// TwinCAT 3 PLC project hydValve
// ProgramVersion: 3.1.4024.0
// libraries:
//   Tc2_Standard, * (Beckhoff Automation GmbH)
//   Tc2_System, * (Beckhoff Automation GmbH)
//   Tc3_Module, * (Beckhoff Automation GmbH)
// project tree:
//   DUTs/ configaracionParammetrs.TcDUT, Staus.TcDUT
//   GVLs/ generalVariable.TcGVL
//   / PlcTask.TcTTO
//   POUs/ accelerationValve.TcPOU, blockMessage.TcPOU, decelerationValve.TcPOU, MAIN.TcPOU, Valve.TcPOU
// real-time tasks:
//   TASK PlcTask: cycle T#10ms, priority 20, ADS port 350

CONFIGURATION hydValve
    RESOURCE PLC ON TwinCAT3
        TASK PlcTask(INTERVAL := T#10ms, PRIORITY := 20);
        PROGRAM MAIN WITH PlcTask : MAIN;
    END_RESOURCE
END_CONFIGURATION

// ---- DUTs/configaracionParammetrs.TcDUT
TYPE configaracionParammetrs :
STRUCT
	CurPosDirMin : REAL := 100; // Minimální proud na solenoid v daném směru [mA]
	CurPosDirMax : REAL := 500; // Maximální proud na solenoid v daném směru [mA]
	CurNegDirMin : REAL := 100; // Minimální proud na solenoid v daném směru [mA]
	CurNegDirMax : REAL := 500; // Maximální proud na solenoid v daném směru [mA]
	RampPosDirUp : INT := 100; // Doba změny z min. na max. otevření v daném směru [ms]
	RampPosDirDown :INT := 100; // Doba změny z max. na min. otevření v daném směru [ms]
	RampNegDirUp : INT := 100; // Doba změny z min. na max. otevření v daném směru [ms]
	RampNegDirDown : INT := 100; // Doba změny z max. na min. otevření v daném směru [ms]
	Deadtime : INT := 5; // Kompenzace setrvačnosti při reverzaci [ms]

END_STRUCT
END_TYPE

// ---- DUTs/Staus.TcDUT
TYPE Staus :
STRUCT
	Standstill : BOOL;	// Oba výstupy jsou na minimu
	Accel : BOOL;	// Jeden z výstupů zrychluje
	Decel : BOOL;	// Jeden z výstupů zpomaluje
	OutPosDirProc : REAL;// Výstup v daném směru [%]
	OutNegDirProc : REAL;// Výstup v daném směru [%]
	bBussy : BOOL;// TRUE je-li FB aktivní (změna na výstupu)
	bDone : BOOL;	// TRUE je-li výstupní hodnota je rovna žádané
	bError : STRING; // Chyba
	nErrorId : INT;// Kód chyby
END_STRUCT
END_TYPE

// ---- GVLs/generalVariable.TcGVL
{attribute 'qualified_only'}
VAR_GLOBAL
	conParammetr : configaracionParammetrs;
	staus : Staus;
END_VAR

// ---- POUs/MAIN.TcPOU
PROGRAM MAIN
VAR
	
	hydraulicValve : Valve;
	enaNegDirB : BOOL := FALSE;
	enaPosDirB : BOOL := FALSE;
	commandSet : REAL := 0;
	//konfiguraParametry : REFERENCE TO configaracionParammetrs  REF=generalVariable.conParammetr;
	OutPosDir : REAL := 0 ;	// Výstup v daném směru [mA]
	OutNegDir : REAL := 0 ;	// Výstup v daném směru [mA]
END_VAR


//hydraulicValve.configaracionParammetr := generalVariable.conParammetr;

hydraulicValve.enableSolenoidControl(poz :=enaPosDirB, neg := enaNegDirB);
hydraulicValve.commandCheck(commandSet);
hydraulicValve();
OutNegDir := hydraulicValve.OutNegDir;
OutPosDir := hydraulicValve.OutPosDir;

END_PROGRAM

// ---- POUs/Valve.TcPOU
FUNCTION_BLOCK Valve
VAR_INPUT
	//configaracionParammetr : configaracionParammetrs;
END_VAR
VAR		
	
	enaNegDir : BOOL := FALSE;
	enaPosDir : BOOL := FALSE;
	command : REAL; // Příkaz -1000 .. 0 .. 1000 [procenta * 10]

	errorDir : BOOL;
	
	currentCommand : REAL := 0;
	prolaz : STRING;
	previousenaNegDir : BOOL; 
	previousenaPosDir : BOOL;
	currentError : BOOL := FALSE; // test error
	
	//command : INT; 
	status : REFERENCE TO Staus REF=generalVariable.staus;
	konfiguraParametry : REFERENCE TO configaracionParammetrs  REF=generalVariable.conParammetr;
	speedRamp : REAL;
	mAcurrentCommand : REAL; 
	mAcommand : REAL;
END_VAR
VAR_OUTPUT
	OutPosDir : REAL := 0 ;	// Výstup v daném směru [mA]
	OutNegDir : REAL := 0 ;	// Výstup v daném směru [mA]
END_VAR

//currentDir := currentDirB(enaNegDir,enaPosDir);
mAcurrentCommand := convertToAnal(ABS(currentCommand*10));
mAcommand :=  convertToAnal(ABS(command*10));

IF (currentCommand = 0) THEN
	OutNegDir := mAcurrentCommand;
	OutPosDir := mAcurrentCommand;
	waitbDeathtime();
	ELSIF enaPosDir > 0 THEN
		OutPosDir := mAcurrentCommand;
		OutNegDir := convertToAnal(0);
		ELSE
			OutNegDir := mAcurrentCommand;
			OutPosDir := convertToAnal(0);
	END_IF;

signalStandstill();
prolaz := 'fb';
IF (currentcommand <> command) THEN
		//nTime := elapsTime(direction := currentDir);
		prolaz := 'različiti';
		currentcommand := rampValve ();
	ELSE	
		Accel_Decel(FALSE, FALSE);
		status.bDone := TRUE;
END_IF;

METHOD PRIVATE Accel_Decel
VAR_INPUT
	a : BOOL;
	b : BOOL;
END_VAR
status.Accel := a;
status.Decel := b;
END_METHOD

METHOD addCommand
VAR_INPUT
	comm : real;
END_VAR
command := comm;	
currentError := FALSE;
errorDir := FALSE;
END_METHOD

METHOD PUBLIC commandCheck
VAR_INPUT
	comm : REAL;
END_VAR
VAR
	
END_VAR
IF not(currentError) THEN
	IF ((comm <= 100) AND (comm >0)) THEN
			IF enaPosDir THEN
				addCommand(comm);
			ELSIF NOT(errorDir) THEN
					errCode(4);
					errorDir := TRUE;
				END_IF
		ELSIF ((comm >= -100) AND (comm < 0)) THEN
				IF enaNegDir THEN
					addCommand(comm);
				ELSIF not(errorDir) THEN
					errCode(3);
					errorDir := TRUE;
				END_IF
				ELSIF comm = 0 THEN
						status.Standstill := 0;
						addCommand(comm);
					ELSIF NOT(errorDir) THEN
					errCode(2);
					errorDir := TRUE;
				END_IF
END_IF
END_METHOD

METHOD PRIVATE convertTo : REAL
VAR_INPUT
	currCommand : REAL;
END_VAR
IF enaPosDir THEN
	convertTo := 100*(currCommand -konfiguraParametry.CurPosDirMin)/(konfiguraParametry.CurPosDirMax - konfiguraParametry.CurPosDirMin);
ELSE
	convertTo := 100*(currCommand -konfiguraParametry.CurNegDirMin)/(konfiguraParametry.CurnegDirMax - konfiguraParametry.CurNegDirMin);
END_IF
END_METHOD

METHOD PROTECTED convertToAnal : REAL
VAR_INPUT
	pCommand : REAL;
END_VAR
IF  enaPosDir THEN
	convertToAnal:= (pCommand * (konfiguraParametry.CurPosDirMax - konfiguraParametry.CurPosDirMin)/1000) + konfiguraParametry.CurPosDirMin;
ELSE
	convertToAnal:= (pCommand * (konfiguraParametry.CurNegDirMax - konfiguraParametry.CurNegDirMin)/1000) + konfiguraParametry.CurNegDirMin;
END_IF
END_METHOD

METHOD PRIVATE elapsTime : REAL
VAR_INPUT
	direction : BOOL;
END_VAR
IF direction THEN
		elapsTime := (konfiguraParametry.CurPosDirMax - konfiguraParametry.CurPosDirMin)/(konfiguraParametry.RampPosDirDown -konfiguraParametry.RampPosDirUp);
	ELSE
		elapsTime := (konfiguraParametry.CurNegDirMax - konfiguraParametry.CurNegDirMin)/(konfiguraParametry.RampNegDirDown -konfiguraParametry.RampNegDirUp);
END_IF
END_METHOD

METHOD PUBLIC enableSolenoidControl
VAR_INPUT
	poz : BOOL;
	neg : BOOL;	
END_VAR
IF (poz AND neg) THEN
	// error 
	errCode(1);
	ELSE
	enaNegDir := neg;
	enaPosDir := poz;
	currentError := FALSE ;
END_IF
END_METHOD

METHOD PRIVATE errCode
VAR_INPUT
	ErrorId : INT; // Kód chyby
END_VAR

CASE ErrorId OF
		1: messageError('muze byt aktivní pouze jedna cívka (PosDir nebo NegDir)');
		2: messageError('hodnot od -100 .. 0 .. 100');
		3: messageError('enable Negativ is False');
		4: messageError('enable Poszitive is False');
		5: messageError('nemuže enable Pos a Neg spolu');
	END_CASE
status.nErrorId := ErrorId;
END_METHOD

METHOD PRIVATE messageError 
VAR_INPUT
	sError :STRING;
END_VAR
IF NOT(currentError) THEN
	status.bError := sError;
	blockMessage(error := sError);
	currentError := TRUE;
END_IF
END_METHOD

METHOD PRIVATE rampTimeCalculate : REAL
VAR_INPUT
	cMax : REAL;
	cMin : REAL;
	rampDirTime : INT;
	delta : real;
END_VAR
rampTimeCalculate := abs((delta * rampDirTime) / (cMax -cMin));
END_METHOD

METHOD PRIVATE rampTimeDown : INT
VAR_INPUT
END_VAR
//RampTimePosDirUp = (configaracionParammetr.CurPosDirMax - configaracionParammetr.CurPosDirMin) / (configaracionParammetr.RampPosDirUp - Deadtime);
END_METHOD

METHOD PRIVATE rampValve : REAL
VAR_INPUT
END_VAR
VAR
	
	delta : REAL;
	rateTime : REAL;
	direction : INT;
END_VAR
prolaz := 'UPAO u rampvalme';
status.Standstill := FALSE;	
IF enaNegDir THEN
	prolaz := 'negTIVNI';
	direction := -1;
	ELSIF enaPosDir THEN
		prolaz := 'pozitivni';
		direction := 1;
END_IF
delta :=  mAcommand - mAcurrentCommand;

IF (currentCommand * command) >= 0 THEN
		// iste znak 
		prolaz := 'isti znak';
					
		IF (delta > 0 ) THEN
			// raste
			prolaz := 'delata veći od 0 ';
			//pitanje da li je dozvola uključena
			
			IF (enaNegDir XOR enaPosDir) THEN
				Accel_Decel(TRUE , FALSE);
				prolaz := 'raste';
				IF (enaPosDir AND command > 0) THEN
						rateTime := rampValveDirection(delta, 1);
					ELSIF (enaNegDir AND command <0) THEN
							rateTime := rampValveDirection(delta, 2);
						ELSE
							command := 0;
				END_IF;
			END_IF;
				mAcurrentCommand := accelerationValve(mAcurrentCommand, mAcommand, rateTime);
		ELSE
			// opada
			prolaz := 'opada';
			Accel_Decel(FALSE , TRUE);
			IF enaNegDir THEN
				rateTime := rampValveDirection(delta, 3);
				ELSE
				rateTime := rampValveDirection(delta, 4);
			END_IF;
			mAcurrentCommand := decelerationValve(mAcurrentCommand, mAcommand, rateTime);
		END_IF;
ELSE
		// različiti znakovi	->	prvo opada
		IF enaNegDir THEN
			rateTime := rampValveDirection(delta, 3);
		ELSE
			rateTime := rampValveDirection(delta, 4);
		END_IF;
		Accel_Decel(FALSE , TRUE);
		mAcurrentCommand := decelerationValve(mAcurrentCommand, 0, rateTime);
END_IF;
	 
delta := convertTo(mAcurrentCommand);
			
rampValve := direction * convertTo(mAcurrentCommand);
END_METHOD

METHOD PRIVATE rampValveDirection : REAL
VAR_INPUT
	delta : REAL;
	i :INT;
END_VAR
CASE i OF
	1:	//Pos  addd
		rampValveDirection := rampTimeCalculate(konfiguraParametry.CurPosDirMax, konfiguraParametry.CurPosDirMin, konfiguraParametry.RampPosDirDown ,delta);
	2: 	//Neg add
		rampValveDirection := rampTimeCalculate(konfiguraParametry.CurNegDirMax, konfiguraParametry.CurNegDirMin, konfiguraParametry.RampNegDirUp ,delta);
	3: 	//pos dec
		rampValveDirection := rampTimeCalculate(konfiguraParametry.CurPosDirMin, konfiguraParametry.CurPosDirMax, konfiguraParametry.RampPosDirDown ,delta);
	4: 	//neg dec
		rampValveDirection := rampTimeCalculate(konfiguraParametry.CurNegDirMin, konfiguraParametry.CurNegDirMax, konfiguraParametry.RampNegDirDown ,delta);
END_CASE
END_METHOD

METHOD signalbBussy : BOOL
VAR_INPUT
END_VAR
END_METHOD

METHOD signalOutDirProc 
VAR_INPUT
	signalOutDirProc : REAL;
END_VAR
VAR_OUTPUT
	OutNegDirProc : REAL;
	OutPosDirProc : real;
END_VAR
signalOutDirProc := command;
IF (signalOutDirProc > 0) THEN
	OutNegDirProc := signalOutDirProc;
	ELSE
		OutPosDirProc := signalOutDirProc;
	END_IF
END_METHOD

METHOD PRIVATE signalStandstill : BOOL
IF (OutPosDir = OutNegDir = 0) THEN
	status.Standstill := TRUE;
	ELSE
		status.Standstill := FALSE;
END_IF
END_METHOD

METHOD PRIVATE speedRampValve 
VAR_INPUT
	i: INT;
END_VAR
// speed Valve transition  Max to min and reverse
CASE i OF
	1 : speedRamp := (konfiguraParametry.CurNegDirMin)/konfiguraParametry.RampNegDirUp;
	2 : speedRamp := (konfiguraParametry.CurNegDirMin)/konfiguraParametry.RampNegDirDown;
	3 : speedRamp := (konfiguraParametry.CurPosDirMin)/konfiguraParametry.RampPosDirUp;
	4 : speedRamp := (konfiguraParametry.CurPosDirMin)/konfiguraParametry.RampPosDirDown;
END_CASE
END_METHOD

METHOD Standstill 
VAR_INPUT
END_VAR
IF (command = 0 ) THEN
	status.Standstill := TRUE;
	blockMessage('Oba výstupy jsou na minimum');
END_IF
END_METHOD

METHOD waitbDeathtime : BOOL
VAR
	delay : TON;
	dTime : TIME;
END_VAR
dTime := INT_TO_TIME(generalVariable.conParammetr.Deadtime);
delay(IN := TRUE, PT:= dtime);
            IF NOT (delay.Q) THEN
                RETURN;
            END_IF;

delay(IN := FALSE);
END_METHOD

END_FUNCTION_BLOCK

// ---- POUs/blockMessage.TcPOU
FUNCTION blockMessage : BOOL
VAR_INPUT
	error : STRING;
END_VAR

ADSLOGSTR(msgCtrlMask := ADSLOG_MSGTYPE_ERROR OR ADSLOG_MSGTYPE_LOG,
	msgFmtStr := error,
	strArg :='');
blockMessage := TRUE;

END_FUNCTION

// ---- POUs/accelerationValve.TcPOU
FUNCTION accelerationValve : REAL
VAR_INPUT
	iCurrent : REAL;
	iTarget : REAL;
	iTime : REAL;
END_VAR
VAR
	delta : REAL;
	time_increment : REAL;
	fbGetCurTaskIdx  : GETCURTASKINDEX;
    nCycleTime       : UDINT;
END_VAR

delta :=  iTarget - iCurrent;

time_increment := ABS(delta/iTime) ;
fbGetCurTaskIdx();
nCycleTime := _TaskInfo[fbGetCurTaskIdx.index].CycleTime;
 
iCurrent := iCurrent + time_increment * nCycleTime;  
IF (iCurrent >= iTarget) THEN
	iCurrent := iTarget;
END_IF
  
 accelerationValve := iCurrent;

END_FUNCTION

// ---- POUs/decelerationValve.TcPOU
FUNCTION decelerationValve : REAL
VAR_INPUT
	iCurrent : REAL;
	iTarget : REAL;
	iTime : REAL;
END_VAR
VAR
	delta : REAL;
	time_increment : REAL;
	fbGetCurTaskIdx  : GETCURTASKINDEX;
     nCycleTime       : UDINT;
END_VAR

delta :=  iTarget - iCurrent ;

time_increment := ABS(delta/iTime) ;
fbGetCurTaskIdx();
nCycleTime := _TaskInfo[fbGetCurTaskIdx.index].CycleTime;
 
iCurrent := iCurrent - time_increment * nCycleTime;  
IF (iCurrent <= iTarget) THEN
	iCurrent := iTarget;
END_IF
decelerationValve := iCurrent ;

END_FUNCTION
